TYPE U_TICKET_LIST_CTRL :
UNION
  stCtrl              : ST_LIST_CTRL;
  byCtrl    AT %I*    : ARRAY[1..SIZEOF(ST_LIST_CTRL)] OF BYTE;
END_UNION
END_TYPE

(* stored: Version 1.1.0.1, ProductVersion 3.1.4026.13
   DUT U_TICKET_LIST_CTRL: Id {8ff08ec9-db69-4d4a-8040-eb6a30ea8a4d} *)
